FUNCTION Camera_Trigger : BOOL
VAR_IN_OUT
	Camera : Cognex_Camera;
END_VAR

IF Camera.CameraState = Camera_State.Idel THEN
	Camera.AcquisitionControl.Clear_Exposure_Complete := TRUE;
	Camera.AcquisitionControl.Acquistion_Trigger := TRUE;
	Camera.CameraState := Camera_State.Jope_Running;
	Camera.JobeState := Job_State.TriggerAck;
	Camera_Trigger := TRUE;
ELSE
	Camera_Trigger := FALSE;
	RETURN;
END_IF

END_FUNCTION

(* stored: Version 1.1.0.1, ProductVersion 3.1.4024.10
   POU Camera_Trigger: Id {ad000b63-df7b-425c-bc71-b905122b4615}, SpecialFunc None *)
